// TwinCAT 3 PLC project PLC1
// ProgramVersion: 3.1.4023.0
// libraries:
//   Tc2_Standard, * (Beckhoff Automation GmbH)
//   Tc2_System, * (Beckhoff Automation GmbH)
//   Tc2_Utilities, * (Beckhoff Automation GmbH)
//   Tc3_IotBase, * (Beckhoff Automation GmbH)
//   Tc3_JsonXml, * (Beckhoff Automation GmbH)
//   Tc3_Module, * (Beckhoff Automation GmbH)
// project tree:
//   DUTs/ E_Query.TcDUT, ST_CurrentSubscription.TcDUT, ST_Data.TcDUT, ST_Homes.TcDUT, ST_TibberPrice.TcDUT, ST_PriceInfo.TcDUT, ST_Result.TcDUT, ST_Viewer.TcDUT
//   GVLs/ GVL.TcGVL
//   / PlcTask.TcTTO
//   POUs/ FB_TibberAPI.TcPOU, MAIN.TcPOU
// real-time tasks:
//   TASK PlcTask: cycle T#10ms, priority 20, ADS port 350

CONFIGURATION PLC1
    RESOURCE PLC ON TwinCAT3
        TASK PlcTask(INTERVAL := T#10ms, PRIORITY := 20);
        PROGRAM MAIN WITH PlcTask : MAIN;
    END_RESOURCE
END_CONFIGURATION

// ---- DUTs/E_Query.TcDUT
{attribute 'qualified_only'}
{attribute 'strict'}
TYPE E_Query :
(
	current := 0,
	today := 1,
	tomorrow := 2,
	all := 3
);
END_TYPE

// ---- DUTs/ST_CurrentSubscription.TcDUT
TYPE ST_CurrentSubscription :
STRUCT
	priceInfo	: ST_PriceInfo;
END_STRUCT
END_TYPE

// ---- DUTs/ST_Data.TcDUT
TYPE ST_Data :
STRUCT
	viewer	: ST_Viewer;
END_STRUCT
END_TYPE

// ---- DUTs/ST_Homes.TcDUT
TYPE ST_Homes :
STRUCT
	currentSubscription	: ST_CurrentSubscription;
END_STRUCT
END_TYPE

// ---- DUTs/ST_TibberPrice.TcDUT
TYPE ST_TibberPrice :
STRUCT
	data	: ST_Data;
END_STRUCT
END_TYPE

// ---- DUTs/ST_PriceInfo.TcDUT
TYPE ST_PriceInfo :
STRUCT
	current		: ST_Result;
	today		: ARRAY [0..23] OF ST_Result;
	tomorrow	: ARRAY [0..23] OF ST_Result;
END_STRUCT
END_TYPE

// ---- DUTs/ST_Result.TcDUT
TYPE ST_Result :
STRUCT
	total    : REAL;
	energy   : REAL;
	tax      : REAL;
	startsAt : STRING;
END_STRUCT
END_TYPE

// ---- DUTs/ST_Viewer.TcDUT
TYPE ST_Viewer :
STRUCT
	homes	: ARRAY[1..GVL.nHomes] OF ST_Homes;
END_STRUCT
END_TYPE

// ---- GVLs/GVL.TcGVL
{attribute 'qualified_only'}
VAR_GLOBAL
	stTibberPrice		: ST_TibberPrice;
END_VAR
VAR_GLOBAL CONSTANT
	nHomes				: UINT := 1;
END_VAR

// ---- POUs/MAIN.TcPOU
PROGRAM MAIN
VAR
	//https://developer.tibber.com/docs/guides/calling-api
	fbTibberClient		: FB_IotHttpClient :=(sHostName := 'api.tibber.com', nHostPort := 443, bKeepAlive := FALSE, stTLS := (bNoServerCertCheck := TRUE));
	fbTibberApi			: FB_TibberApi;
	// Tibber Demo Token: 5K4MVS-OjfWhK_4yrjOlFe1F6kJXPVf7eQYggo8ebAE
	sToken				: STRING := '5K4MVS-OjfWhK_4yrjOlFe1F6kJXPVf7eQYggo8ebAE';
	eQuery				: E_Query;
	bRun				: BOOL;
	bError				: BOOL;
	bBusy				: BOOL;
	nStatus				: UINT;
END_VAR

IF fbTibberClient.bConfigured THEN
	fbTibberApi(
		bSend:= bRun, 
		fbClient:= fbTibberClient, 
		pTibberPrice:= ADR(GVL.stTibberPrice), 
		nSize:= SIZEOF(GVL.stTibberPrice),
		sToken:= sToken,
		eQuery:= eQuery,
		bBusy=> bBusy, 
		bError=> bError,
		nStatus=> nStatus );
END_IF
fbTibberClient.Execute();

END_PROGRAM

// ---- POUs/FB_TibberAPI.TcPOU
FUNCTION_BLOCK FB_TibberAPI
//Tested and works with 4024.22 4024.29 4024.32 4024.35
//Will not work with any 4022. 4024.7 may also not work.
//Based on the Beckhoff Postman POST example: https://infosys.beckhoff.com/content/1033/tf6760_tc3_iot_https_rest/7876792971.html?id=8531523618449441037
VAR_INPUT
    bSend				: BOOL;
	pTibberPrice		: PVOID;
	nSize				: UINT;
	sToken				: STRING;
	eQuery				: E_Query;
END_VAR
VAR_IN_OUT
    fbClient            : FB_IotHttpClient;
END_VAR
VAR_OUTPUT
    bBusy               : BOOL;
    bError              : BOOL;
	nStatus				: UINT;
END_VAR
VAR
    fbRequest           : FB_IotHttpRequest;
	fbHeader            : FB_IotHttpHeaderFieldMap;
    fbJson              : FB_JsonDomParser;
	fbJsonDataType		: FB_JsonReadWriteDataType;
	RisingEdge          : R_TRIG; 
    sContent            : STRING (4095);
	sContentReceive		: STRING (6143);
    nErrCount           : UDINT;
	nState              : UDINT;
END_VAR

RisingEdge(CLK:= bSend);
CASE nState OF
0:
    IF RisingEdge.Q THEN
		sToken := CONCAT('Bearer	', sToken);
		fbHeader.AddField('Authorization', sToken, FALSE);
		fbRequest.sContentType := 'application/json; charset=utf-8';
		sContent := M_QueryType(eQuery := eQuery);
        IF fbRequest.SendRequest(sUri:= '/v1-beta/gql/', fbClient:= fbClient, eRequestType:= ETcIotHttpRequestType.HTTP_POST, pContent:= ADR(sContent), nContentSize:= LEN2(ADR(sContent)), fbHeader:=fbHeader) THEN
            nState:= 1;
            bBusy:= TRUE;
            bError:= FALSE;
        END_IF
    END_IF
1:	
	IF NOT fbRequest.bBusy THEN
		bError:= TRUE;
		IF NOT fbRequest.bError THEN				 					
			IF fbRequest.GetContent(pContent:= ADR(sContentReceive), nContentSize:= SIZEOF(sContentReceive), bSetNullTermination:= TRUE) AND fbRequest.nStatusCode >= 200 AND fbRequest.nStatusCode < 300 THEN
					IF fbJsonDataType.SetSymbolFromJson(sContentReceive, 'ST_TibberPrice', nSize, pTibberPrice) THEN
						bError:= FALSE;
					END_IF				
			END_IF				
		END_IF
		nState:= 0;
		nStatus := fbRequest.nStatusCode;
		bBusy:= FALSE;
		IF bError THEN
			nErrCount:= nErrCount+1;
		END_IF		
	END_IF  	
END_CASE

METHOD M_QueryType : STRING (4095)
VAR_INPUT
	eQuery		: E_Query;
END_VAR
CASE eQuery OF
	E_Query.current:
		M_QueryType:= '{ "query": "{viewer {homes {currentSubscription{priceInfo{current{total energy tax startsAt }}}}}}" }';
	E_Query.today:
		M_QueryType:= '{ "query": "{viewer {homes {currentSubscription {priceInfo {today {total energy tax startsAt }}}}}}" }';
	E_Query.tomorrow:
		M_QueryType:= '{ "query": "{viewer {homes {currentSubscription {priceInfo {tomorrow {total energy tax startsAt }}}}}}" }';
	E_Query.all:
		M_QueryType:= '{ "query": "{viewer {homes{currentSubscription {priceInfo {current {total energy tax startsAt}today {total energy tax startsAt}tomorrow {total energy tax startsAt }}}}}}" }';
END_CASE
END_METHOD

END_FUNCTION_BLOCK
